(* IEC 61131-3 sources: plc_generation_empirical_study/datasets/task_bank_c04_reverse_runtime_v0_2/tasks/C04_R24_lean_composite, 2 files *)

(* ---- interface.st ---- *)
FUNCTION_BLOCK C04_R24_lean_composite
VAR_INPUT
    A_Ch1 : BOOL;
    A_Ch2 : BOOL;
    A_Ch3 : BOOL;
    A_AutoMode : BOOL;
    A_AutoRequest : BOOL;
    A_ManualRequest : BOOL;
    A_BypassRequest : BOOL;
    A_BypassPermit : BOOL;
    A_SafetyOK : BOOL;
    A_Reset : BOOL;
    B_Button : BOOL;
    B_Enable : BOOL;
    B_Reset : BOOL;
    SubsystemBEnable : BOOL;
    CrossReset : BOOL;
END_VAR
VAR_OUTPUT
    A_RunPermit : BOOL;
    A_Degraded : BOOL;
    A_BypassActive : BOOL;
    A_Blocked : BOOL;
    B_State : BOOL;
    B_AcceptedPulse : BOOL;
    CrossReady : BOOL;
    CrossBlocked : BOOL;
END_VAR
END_FUNCTION_BLOCK

(* ---- reference.st ---- *)
FUNCTION_BLOCK C04_R24_lean_composite
VAR_INPUT
    A_Ch1 : BOOL;
    A_Ch2 : BOOL;
    A_Ch3 : BOOL;
    A_AutoMode : BOOL;
    A_AutoRequest : BOOL;
    A_ManualRequest : BOOL;
    A_BypassRequest : BOOL;
    A_BypassPermit : BOOL;
    A_SafetyOK : BOOL;
    A_Reset : BOOL;
    B_Button : BOOL;
    B_Enable : BOOL;
    B_Reset : BOOL;
    SubsystemBEnable : BOOL;
    CrossReset : BOOL;
END_VAR
VAR_OUTPUT
    A_RunPermit : BOOL;
    A_Degraded : BOOL;
    A_BypassActive : BOOL;
    A_Blocked : BOOL;
    B_State : BOOL;
    B_AcceptedPulse : BOOL;
    CrossReady : BOOL;
    CrossBlocked : BOOL;
END_VAR
VAR
    A_SelectedRequest : BOOL;
    A_VoteOK : BOOL;
    A_AnyChannel : BOOL;
    A_Unanimous : BOOL;
    B_PrevButton : BOOL := FALSE;
END_VAR

A_SelectedRequest := (A_AutoMode AND A_AutoRequest) OR ((NOT A_AutoMode) AND A_ManualRequest);
A_VoteOK := (A_Ch1 AND A_Ch2) OR (A_Ch1 AND A_Ch3) OR (A_Ch2 AND A_Ch3);
A_AnyChannel := A_Ch1 OR A_Ch2 OR A_Ch3;
A_Unanimous := (A_Ch1 AND A_Ch2 AND A_Ch3) OR ((NOT A_Ch1) AND (NOT A_Ch2) AND (NOT A_Ch3));
IF A_Reset AND (NOT A_AutoRequest) AND (NOT A_ManualRequest) THEN
    A_BypassActive := FALSE;
ELSIF (NOT A_AutoMode) AND A_BypassRequest AND A_BypassPermit AND A_SafetyOK AND A_AnyChannel THEN
    A_BypassActive := TRUE;
END_IF;
A_RunPermit := A_SelectedRequest AND A_SafetyOK AND (A_VoteOK OR A_BypassActive);
A_Degraded := A_RunPermit AND ((NOT A_Unanimous) OR A_BypassActive);
A_Blocked := A_SelectedRequest AND (NOT A_RunPermit);

IF CrossReset THEN
    CrossReady := FALSE;
ELSIF A_RunPermit THEN
    CrossReady := TRUE;
END_IF;
CrossBlocked := SubsystemBEnable AND (NOT CrossReady);

IF SubsystemBEnable AND CrossReady THEN
    B_AcceptedPulse := FALSE;
    IF B_Reset THEN
        B_State := FALSE;
    ELSIF B_Enable AND B_Button AND (NOT B_PrevButton) THEN
        B_State := NOT B_State;
        B_AcceptedPulse := TRUE;
    END_IF;
    B_PrevButton := B_Button;
ELSE
    B_State := FALSE;
    B_AcceptedPulse := FALSE;
END_IF;

END_FUNCTION_BLOCK
